TYPE Inner_conveyor :
STRUCT
	belt	: ARRAY[0..2] OF Belt;
	valve	: ARRAY[0..2] OF Valve;
	rfid	: ARRAY[0..1] OF RFID;
	photo_sensor	: ARRAY[0..5] OF BOOL;
END_STRUCT
END_TYPE

(* stored: Version 1.1.0.1, ProductVersion 3.1.4024.12
   DUT Inner_conveyor: Id {f5c0ba46-6e55-43a2-9b5a-0ab2105d475b} *)
